{attribute 'linkalways'} 
{attribute 'no_explicit_call' := 'This FB is a CLASS and must be accessed using methods or properties'}
{attribute 'enable_dynamic_creation'}
FUNCTION_BLOCK MiddlewareStack
VAR
	InitialHandler : I_Middleware;
END_VAR

METHOD PUBLIC Handle
VAR_INPUT
	Request : I_Request;
	Response : I_ServerResponse;
END_VAR
IF initialHandler = 0 THEN
	RETURN;
END_IF

initialHandler.Handle(Request, Response);
END_METHOD

METHOD PUBLIC Use
VAR_INPUT
	Handler : I_Middleware;
END_VAR
VAR
	currentHandler : I_Middleware;
END_VAR;
IF initialHandler = 0 THEN
	initialHandler := Handler;
	RETURN;
END_IF

currentHandler := InitialHandler;

WHILE currentHandler.NextMiddleware <> 0 DO
	currentHandler := currentHandler.NextMiddleware;
END_WHILE

currentHandler.NextMiddleware := Handler;
END_METHOD

END_FUNCTION_BLOCK

(* stored: Version 1.1.0.1, ProductVersion 3.1.4024.12
   POU MiddlewareStack: Id {d4b384e4-9cd9-4072-8cb6-38e686023b60}, SpecialFunc None
   Method Handle: Id {0b963707-e7d9-4ad3-aab7-3ea5ae7fa1bf}
   Method Use: Id {120fb1d4-0605-4cc8-bc81-f8ffeb9c2263} *)
